{attribute 'qualified_only'}
{attribute 'strict'}
TYPE E_Step :
(
	
	(* special steps *)
	NoStep		:=	-32767,
	Unknown		:=	-32000,
	
	(* Not Enabled or Errors*)
	NeOrError	:=	-990,
	
	(* Stop *)
	Stop		:=	0,
	
	(* CSL's steps *)
	Start		:= 	100,
	Measuring	:= 	110,
	Processing	:= 	120,
	conveyor	:= 	130,
	waiting		:= 	140,
	piston		:= 	150,
	
	Stopping	:=	900
);
END_TYPE

(* stored: Version 1.1.0.1, ProductVersion 3.1.4024.12
   DUT E_Step: Id {6d3f40d7-f503-4f78-b3a8-51bf47e61ef9} *)
